PROGRAM MAIN
VAR
	

mCTCInSpeedSuggested : ARRAY[0..149] OF DINT;
mCTCInAuthority : ARRAY[0..149] OF DINT;
mCTCInMaintenanceMode : ARRAY[0..149] OF DINT;
mCTCInSwitchPosition : ARRAY[0..149] OF DINT;

mTrackInMaintenanceMode : ARRAY[0..149] OF DINT;
mTrackInSwitchPosition : ARRAY[0..149] OF DINT;
mTrackInOccupancy : ARRAY[0..149] OF DINT;
mTrackInCrossing : ARRAY[0..149] OF DINT;
mTrackInRightTransit : ARRAY[0..149] OF DINT;
mTrackInLeftTransit : ARRAY[0..149] OF DINT;
mTrackOutSpeedSuggested : ARRAY[0..149] OF DINT;
mTrackOutAuthority : ARRAY[0..149] OF DINT;
mOutMaintenanceMode : ARRAY[0..149] OF DINT;
mOutSwitchPosition : ARRAY[0..149] OF DINT;
mOutOccupancy : ARRAY[0..149] OF DINT;
mOutCrossing : ARRAY[0..149] OF DINT;
mOutRightTransit : ARRAY[0..149] OF DINT;
mOutLeftTransit : ARRAY[0..149] OF DINT;

mPLC2MismatchCounter : DINT :=0;
mPLC3MismatchCounter : DINT :=0;
mPLC2MismatchFlag : BOOL := 0;
mPLC3MismatchFlag : BOOL := 0;


	inc1: INT;
END_VAR

FOR inc1 := 0 TO 149 DO

mCTCInSpeedSuggested[inc1] := GVL.mInFromCTC[inc1+0];
mCTCInAuthority[inc1] := GVL.mInFromCTC[inc1+150];
mCTCInMaintenanceMode[inc1] := GVL.mInFromCTC[inc1+300];
mCTCInSwitchPosition[inc1] := GVL.mInFromCTC[inc1+450];

mOutMaintenanceMode[inc1] := GVL.mInFromTrack[inc1+0];
mOutSwitchPosition[inc1] := GVL.mInFromTrack[inc1+150];
mOutOccupancy[inc1] := GVL.mInFromTrack[inc1+300];
mOutCrossing[inc1] := GVL.mInFromTrack[inc1+450];
mOutRightTransit[inc1] := GVL.mInFromTrack[inc1+600];
mOutLeftTransit[inc1] := GVL.mInFromTrack[inc1+750];

END_FOR


FOR inc1 := 0 TO 149 DO

IF GVL.mWriteEnable = 1 THEN
GVL.mOutToTrack[inc1+0] := mTrackOutSpeedSuggested[inc1];
GVL.mOutToTrack[inc1+150] := mTrackOutAuthority[inc1]; 
GVL.mOutToTrack[inc1+300] := mOutMaintenanceMode[inc1];
GVL.mOutToTrack[inc1+450] := mOutSwitchPosition[inc1] ;
GVL.mOutToTrack[inc1+600] := mOutOccupancy[inc1];
GVL.mOutToTrack[inc1+750] := mOutCrossing[inc1];
GVL.mOutToTrack[inc1+900] := mOutRightTransit[inc1];
GVL.mOutToTrack[inc1+1050] := mOutLeftTransit[inc1];

GVL.mOutToCTC[inc1+0] := mOutMaintenanceMode[inc1];
GVL.mOutToCTC[inc1+150] := mOutSwitchPosition[inc1] ;
GVL.mOutToCTC[inc1+300] := mOutOccupancy[inc1];
GVL.mOutToCTC[inc1+450] := mOutCrossing[inc1];
GVL.mOutToCTC[inc1+600] := mOutRightTransit[inc1];
GVL.mOutToCTC[inc1+750] := mOutLeftTransit[inc1];

IF GVL.mOutToTrack[inc1+0] <> GVL.mPLC2TrackWrites[inc1+0] THEN
    mPLC2MismatchFlag := mPLC2MismatchFlag OR 1;
	END_IF
IF GVL.mOutToTrack[inc1+150] <> GVL.mPLC2TrackWrites[inc1+150] THEN
    mPLC2MismatchFlag := mPLC2MismatchFlag OR 1;
	END_IF
IF GVL.mOutToTrack[inc1+300] <> GVL.mPLC2TrackWrites[inc1+300] THEN
    mPLC2MismatchFlag := mPLC2MismatchFlag OR 1;
	END_IF
IF GVL.mOutToTrack[inc1+450] <> GVL.mPLC2TrackWrites[inc1+450] THEN
    mPLC2MismatchFlag := mPLC2MismatchFlag OR 1;
	END_IF
IF GVL.mOutToTrack[inc1+600] <> GVL.mPLC2TrackWrites[inc1+600] THEN
    mPLC2MismatchFlag := mPLC2MismatchFlag OR 1;
	END_IF
IF GVL.mOutToTrack[inc1+750] <> GVL.mPLC2TrackWrites[inc1+750] THEN
    mPLC2MismatchFlag := mPLC2MismatchFlag OR 1;
	END_IF
IF GVL.mOutToTrack[inc1+900] <> GVL.mPLC2TrackWrites[inc1+900] THEN
    mPLC2MismatchFlag := mPLC2MismatchFlag OR 1;
	END_IF
IF GVL.mOutToTrack[inc1+1050] <> GVL.mPLC2TrackWrites[inc1+1050] THEN
    mPLC2MismatchFlag := mPLC2MismatchFlag OR 1;
	END_IF

IF GVL.mOutToCTC[inc1+0] <> GVL.mPLC2CTCWrites[inc1+0] THEN
    mPLC2MismatchFlag := mPLC2MismatchFlag OR 1;
	END_IF
IF GVL.mOutToCTC[inc1+150] <> GVL.mPLC2CTCWrites[inc1+150] THEN
    mPLC2MismatchFlag := mPLC2MismatchFlag OR 1;
	END_IF
IF GVL.mOutToCTC[inc1+300] <> GVL.mPLC2CTCWrites[inc1+300] THEN
    mPLC2MismatchFlag := mPLC2MismatchFlag OR 1;
	END_IF
IF GVL.mOutToCTC[inc1+450] <> GVL.mPLC2CTCWrites[inc1+450] THEN
    mPLC2MismatchFlag := mPLC2MismatchFlag OR 1;
	END_IF
IF GVL.mOutToCTC[inc1+600] <> GVL.mPLC2CTCWrites[inc1+600] THEN
    mPLC2MismatchFlag := mPLC2MismatchFlag OR 1;
	END_IF
IF GVL.mOutToCTC[inc1+750] <> GVL.mPLC2CTCWrites[inc1+750] THEN
    mPLC2MismatchFlag := mPLC2MismatchFlag OR 1;
	END_IF

IF GVL.mOutToTrack[inc1+0] <> GVL.mPLC3TrackWrites[inc1+0] THEN
    mPLC3MismatchFlag := mPLC3MismatchFlag OR 1;
	END_IF
IF GVL.mOutToTrack[inc1+150] <> GVL.mPLC3TrackWrites[inc1+150] THEN
    mPLC3MismatchFlag := mPLC3MismatchFlag OR 1;
	END_IF
IF GVL.mOutToTrack[inc1+300] <> GVL.mPLC3TrackWrites[inc1+300] THEN
    mPLC3MismatchFlag := mPLC3MismatchFlag OR 1;
	END_IF
IF GVL.mOutToTrack[inc1+450] <> GVL.mPLC3TrackWrites[inc1+450] THEN
    mPLC3MismatchFlag := mPLC3MismatchFlag OR 1;
	END_IF
IF GVL.mOutToTrack[inc1+600] <> GVL.mPLC3TrackWrites[inc1+600] THEN
    mPLC3MismatchFlag := mPLC3MismatchFlag OR 1;
	END_IF
IF GVL.mOutToTrack[inc1+750] <> GVL.mPLC3TrackWrites[inc1+750] THEN
    mPLC3MismatchFlag := mPLC3MismatchFlag OR 1;
	END_IF
IF GVL.mOutToTrack[inc1+900] <> GVL.mPLC3TrackWrites[inc1+900] THEN
    mPLC3MismatchFlag := mPLC3MismatchFlag OR 1;
	END_IF
IF GVL.mOutToTrack[inc1+1050] <> GVL.mPLC3TrackWrites[inc1+1050] THEN
    mPLC3MismatchFlag := mPLC3MismatchFlag OR 1;
	END_IF

IF GVL.mOutToCTC[inc1+0] <> GVL.mPLC3CTCWrites[inc1+0] THEN
    mPLC3MismatchFlag := mPLC3MismatchFlag OR 1;
	END_IF
IF GVL.mOutToCTC[inc1+150] <> GVL.mPLC3CTCWrites[inc1+150] THEN
    mPLC3MismatchFlag := mPLC3MismatchFlag OR 1;
	END_IF
IF GVL.mOutToCTC[inc1+300] <> GVL.mPLC3CTCWrites[inc1+300] THEN
    mPLC3MismatchFlag := mPLC3MismatchFlag OR 1;
	END_IF
IF GVL.mOutToCTC[inc1+450] <> GVL.mPLC3CTCWrites[inc1+450] THEN
    mPLC3MismatchFlag := mPLC3MismatchFlag OR 1;
	END_IF
IF GVL.mOutToCTC[inc1+600] <> GVL.mPLC2CTCWrites[inc1+600] THEN
    mPLC3MismatchFlag := mPLC3MismatchFlag OR 1;
	END_IF
IF GVL.mOutToCTC[inc1+750] <> GVL.mPLC3CTCWrites[inc1+750] THEN
    mPLC3MismatchFlag := mPLC3MismatchFlag OR 1;
	END_IF
ELSE
GVL.mOutToTrack[inc1+0] := 0;
GVL.mOutToTrack[inc1+150] := 0; 
GVL.mOutToTrack[inc1+300] := 0;
GVL.mOutToTrack[inc1+450] := 0 ;
GVL.mOutToTrack[inc1+600] := 0;
GVL.mOutToTrack[inc1+750] := 0;
GVL.mOutToTrack[inc1+900] := 0;
GVL.mOutToTrack[inc1+1050] := 0;

GVL.mOutToCTC[inc1+0] := 0;
GVL.mOutToCTC[inc1+150] := 0;
GVL.mOutToCTC[inc1+300] := 0;
GVL.mOutToCTC[inc1+450] := 0;
GVL.mOutToCTC[inc1+600] := 0;
GVL.mOutToCTC[inc1+750] := 0;
END_IF
END_FOR


(*
IF mPLC2MismatchFlag = 1 THEN
    mPLC2MismatchCounter := mPLC2MismatchCounter + 1;
ELSE
    mPLC2MismatchCounter := 0;
END_IF
IF mPLC3MismatchFlag = 1 THEN
    mPLC3MismatchCounter := mPLC3MismatchCounter + 1;
ELSE
    mPLC3MismatchCounter := 0;
END_IF


IF mPLC2MismatchCounter > 10 THEN
    mPLC2MismatchFlag := 1;
    GVL.mPLC2Failure := 1;
END_IF
IF mPLC3MismatchCounter > 10 THEN
    mPLC3MismatchFlag := 1;
    GVL.mPLC3Failure := 1;
END_IF

IF GVL.mPLC2Failure AND GVL.mPLC3Failure Then
    GVL.mWriteEnable := 0;
END_IF;
*)

END_PROGRAM

(* stored: Version 1.1.0.1, ProductVersion 3.1.4024.11
   POU MAIN: Id {4c8b3e77-e4d8-438f-9dd4-fa42d08617c7}, SpecialFunc None *)
